FUNCTION F_ReadRobotPosition : REAL
VAR_INPUT
	IN_Upper		: WORD; //The Upper 16 Bits data (1st WORD) from Full 32 Bits Data(DWORD)
	IN_Lower		: WORD; //The Lower 16 Bits data (2st WORD) from Full 32 Bits Data(DWORD)
END_VAR
VAR
	d_Input : DWORD;
	i_Input : REAL;
END_VAR

// IN_Upper is WORD from KUKA EIP
//d_Input = DWORD
//INSERT WORD INTO DWORD
// SHL Shift Left 16 bit of data + Lower 16 bit of data 
// Convert DWORD to REAL 

d_Input :=  IN_Upper;
d_Input := SHL(d_Input,16) + IN_Lower;
i_Input:= TO_REAL(DWORD_TO_DINT(d_Input));
F_ReadRobotPosition := (i_Input/1000);

END_FUNCTION

(* stored: Version 1.1.0.1, ProductVersion 3.1.4024.11
   POU F_ReadRobotPosition: Id {d09d1508-98a7-4d6a-bc37-558579fe2899}, SpecialFunc None *)
